(* This function block impelemets Interlock for Agilent Turbo Vent Valve Normally Open*)
FUNCTION_BLOCK FB_TurbVentvalve_NO
VAR_OUTPUT
    {attribute 'pytmc' :=' pv:'}
    q_stValve : ST_VCC_NO;
END_VAR
VAR_INPUT
    i_stPTM	: ST_AgilentPTM; //Agilent Turbo Pump
END_VAR
VAR
    tofTmr 		: 	TOF;

    (*Output*)
    q_xCLS_DO AT%Q* : BOOL;
END_VAR

(*If the turbo is on, you cannot open the valve. In order to open the valve, you have to allow the turbopump
 to have already been turned off for 2 minutes and you have to press the open button on the vent valve

If the code looks confusing please use a truth table to verify*)

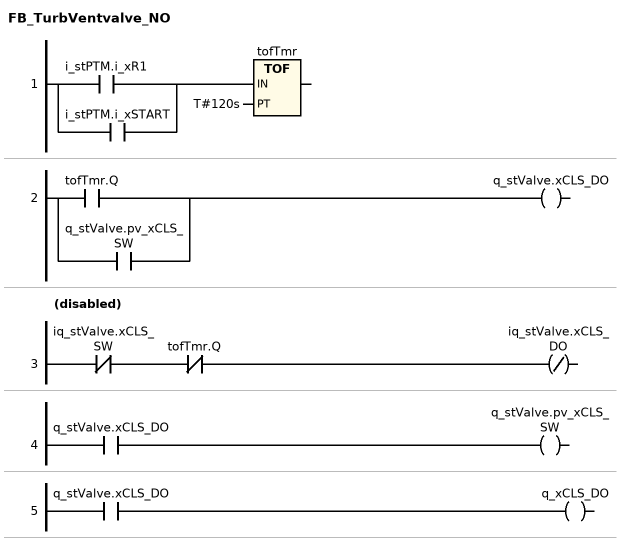
// NETWORK 1
tofTmr(IN := i_stPTM.i_xR1 OR i_stPTM.i_xSTART, PT := T#120s); // TOF

// NETWORK 2
q_stValve.xCLS_DO := tofTmr.Q OR q_stValve.pv_xCLS_SW;

// NETWORK 3 (disabled)
// iq_stValve.xCLS_DO := NOT (NOT iq_stValve.xCLS_SW AND NOT tofTmr.Q);

// NETWORK 4
q_stValve.pv_xCLS_SW := q_stValve.xCLS_DO;

// NETWORK 5
q_xCLS_DO := q_stValve.xCLS_DO;

ACTION ACT_IO:
(*outputs*)
q_xCLS_DO:= q_stValve.xCLS_DO;
END_ACTION

METHOD M_Close : BOOL
VAR_INPUT
        close:BOOL; //True to CLose, False to OPEN
END_VAR
This^.q_stValve.pv_xCLS_SW :=Close;
END_METHOD

END_FUNCTION_BLOCK

(* stored: Version 1.1.0.1
   POU FB_TurbVentvalve_NO: Id {13f6dcdf-6eaf-4953-b8b2-2ecf46768828}, SpecialFunc None
   Action ACT_IO: Id {10c4199c-404d-42f2-a93b-68c98ae69b96}
   Method M_Close: Id {f952aee4-b56f-449f-acf0-34ee976bf562} *)
